// TwinCAT 3 PLC project VersionLib
// Title: VersionLib
// Company: FactoryAutomation
// Author: Filippo Boido
// ProjectVersion: 1.2.0.2
// ProgramVersion: 3.1.4023.0
// libraries:
//   Tc2_Standard, * (Beckhoff Automation GmbH)
//   Tc2_System, * (Beckhoff Automation GmbH)
//   Tc3_Module, * (Beckhoff Automation GmbH)
//   VersionLib, * (FactoryAutomation)
// project tree:
//   / CheckVersion.TcPOU, GetBuild.TcPOU, GetMajor.TcPOU, GetMinor.TcPOU, GetRevision.TcPOU, Version.TcGVL

// ---- Version.TcGVL
{attribute 'qualified_only'}
VAR_GLOBAL CONSTANT
	Major : UINT;
	Minor : UINT;
	Revision : UINT;
	Build : UINT;
END_VAR

// ---- CheckVersion.TcPOU
FUNCTION CheckVersion : BOOL
VAR_INPUT
	Major : UINT;
	Minor : UINT;
	Revision : UINT;
	Build : UINT;
END_VAR
VAR
END_VAR

IF Major = Version.Major
 AND Minor = Version.Minor
 AND Revision = Version.Revision
 AND Build = Version.Build
THEN
	CheckVersion := TRUE;
END_IF

END_FUNCTION

// ---- GetBuild.TcPOU
FUNCTION GetBuild : UINT
VAR_INPUT
END_VAR
VAR
END_VAR

GetBuild := Version.Build;

END_FUNCTION

// ---- GetMajor.TcPOU
FUNCTION GetMajor : UINT
VAR_INPUT
END_VAR
VAR
END_VAR

GetMajor := Version.Major;

END_FUNCTION

// ---- GetMinor.TcPOU
FUNCTION GetMinor : UINT
VAR_INPUT
END_VAR
VAR
END_VAR

GetMinor := Version.Minor;

END_FUNCTION

// ---- GetRevision.TcPOU
FUNCTION GetRevision : UINT
VAR_INPUT
END_VAR
VAR
END_VAR

GetRevision := Version.Revision;

END_FUNCTION
